(* CODESYS project 2ndTest

Project tree, tasks and I/O mapping:
  Device : XV300, Eaton Automation, version 3.5.17.30
    application Application
      libraries: Standard, 3.5.17.0 (System)
      task MainTask (cyclic, interval t#10ms, priority 1) calls PLC_PRG
      program PLC_PRG [ST]
*)

// Device/Application/PLC_PRG
PROGRAM PLC_PRG
VAR
	i: INT;
END_VAR

i:=i+1;

END_PROGRAM
